{attribute 'GeneratedUsingTerminal: EK1100-0000-0018'}
{attribute addProperty BoxType "EK1100-0000-0018"}
{attribute addProperty Id "Beckhoff_EJ7xxxEK1122Beckhoff_EJ7xxxEK1122_3A43B2222A_0001_EJ7031_0000_0026EJ7031_31AD1E8938A_0002_EJ7037_0000_0020EJ7037_B6E6359B46A_0003_EJ7041_0052_0016EJ7041_31AD1E8938A_0004_EJ7047_0000_0018EJ7047_B6E6359B46A_0005_EJ7047_0000_0019EJ7047_B6E6359B46A_0006_EJ7047_0000_0020EJ7047_B6E6359B46A_0007_EJ7342_0000_0019EJ7342_A970B60778A_0008_EJ7342_0000_0020EJ7342_A970B60778A_0009_EJ7211_0010_0026EJ7211_91DE43F025A_0010_EJ7211_0010_0027EJ7211_91DE43F025A_0011_EJ7211_0010_0028EJ7211_91DE43F025A_0012_EJ7211_0010_0029EJ7211_91DE43F025A_0013_EJ7211_0010_0030EJ7211_0985306B26A_0014_EJ7211_0010_0031EJ7211_0985306B26A_0015_EJ7211_0010_0032EJ7211_0985306B26A_0016_EJ7211_0011_0026EJ7211_24495B2825A_0017_EJ7211_0011_0027EJ7211_24495B2825A_0018_EJ7211_0011_0028EJ7211_24495B2825A_0019_EJ7211_0011_0029EJ7211_24495B2825A_0020_EJ7211_0011_0030EJ7211_24495B2825A_0021_EJ7211_0011_0031EJ7211_24495B2825A_0022_EJ7211_0011_0032EJ7211_24495B2825A_0023_EJ7211_9414_0029EJ7211_91DE43F025A_0024_EJ7211_9414_0030EJ7211_49D18A3927A_0025_EJ7211_9414_0031EJ7211_49D18A3927A_0026_EJ7211_9414_0032EJ7211_49D18A3927A_0027_EJ7211_9415_0029EJ7211_24495B2825A_0028_EJ7211_9415_0030EJ7211_24495B2825A_0029_EJ7211_9415_0031EJ7211_24495B2825A_0030_EJ7211_9415_0032EJ7211_24495B2825A_0031_EJ7334_0008_0016EJ7334_074992E952A_0032_EJ7411_0000_0018EJ7411_D6A8D49830"}
{attribute addProperty CRC "2174237961"}
{attribute addProperty Size "1059"}
TYPE Beckhoff_EJ7xxx_81983D09 EXTENDS EK1100_1FC0878B :
STRUCT
	{attribute addProperty Name "Beckhoff_EJ7xxxEK1122"}
	{attribute addProperty PreviousPort "Beckhoff EJ7xxx : B"}
	Beckhoff_EJ7xxxEK1122 : Beckhoff_EJ7xxxEK1122_3A43B222;
	{attribute addProperty Name "A_0001_EJ7031_0000_0026"}
	{attribute addProperty PreviousPort "Beckhoff EJ7xxxEK1122 : C"}
	A_0001_EJ7031_0000_0026 : EJ7031_31AD1E89;
	{attribute addProperty Name "A_0002_EJ7037_0000_0020"}
	{attribute addProperty PreviousPort "A_0001(EJ7031-0000-0026) : B"}
	A_0002_EJ7037_0000_0020 : EJ7037_B6E6359B;
	{attribute addProperty Name "A_0003_EJ7041_0052_0016"}
	{attribute addProperty PreviousPort "A_0002(EJ7037-0000-0020) : B"}
	A_0003_EJ7041_0052_0016 : EJ7041_31AD1E89;
	{attribute addProperty Name "A_0004_EJ7047_0000_0018"}
	{attribute addProperty PreviousPort "A_0003(EJ7041-0052-0016) : B"}
	A_0004_EJ7047_0000_0018 : EJ7047_B6E6359B;
	{attribute addProperty Name "A_0005_EJ7047_0000_0019"}
	{attribute addProperty PreviousPort "A_0004(EJ7047-0000-0018) : B"}
	A_0005_EJ7047_0000_0019 : EJ7047_B6E6359B;
	{attribute addProperty Name "A_0006_EJ7047_0000_0020"}
	{attribute addProperty PreviousPort "A_0005(EJ7047-0000-0019) : B"}
	A_0006_EJ7047_0000_0020 : EJ7047_B6E6359B;
	{attribute addProperty Name "A_0007_EJ7342_0000_0019"}
	{attribute addProperty PreviousPort "A_0006(EJ7047-0000-0020) : B"}
	A_0007_EJ7342_0000_0019 : EJ7342_A970B607;
	{attribute addProperty Name "A_0008_EJ7342_0000_0020"}
	{attribute addProperty PreviousPort "A_0007(EJ7342-0000-0019) : B"}
	A_0008_EJ7342_0000_0020 : EJ7342_A970B607;
	{attribute addProperty Name "A_0009_EJ7211_0010_0026"}
	{attribute addProperty PreviousPort "A_0008(EJ7342-0000-0020) : B"}
	A_0009_EJ7211_0010_0026 : EJ7211_91DE43F0;
	{attribute addProperty Name "A_0010_EJ7211_0010_0027"}
	{attribute addProperty PreviousPort "A_0009(EJ7211-0010-0026) : B"}
	A_0010_EJ7211_0010_0027 : EJ7211_91DE43F0;
	{attribute addProperty Name "A_0011_EJ7211_0010_0028"}
	{attribute addProperty PreviousPort "A_0010(EJ7211-0010-0027) : B"}
	A_0011_EJ7211_0010_0028 : EJ7211_91DE43F0;
	{attribute addProperty Name "A_0012_EJ7211_0010_0029"}
	{attribute addProperty PreviousPort "A_0011(EJ7211-0010-0028) : B"}
	A_0012_EJ7211_0010_0029 : EJ7211_91DE43F0;
	{attribute addProperty Name "A_0013_EJ7211_0010_0030"}
	{attribute addProperty PreviousPort "A_0012(EJ7211-0010-0029) : B"}
	A_0013_EJ7211_0010_0030 : EJ7211_0985306B;
	{attribute addProperty Name "A_0014_EJ7211_0010_0031"}
	{attribute addProperty PreviousPort "A_0013(EJ7211-0010-0030) : B"}
	A_0014_EJ7211_0010_0031 : EJ7211_0985306B;
	{attribute addProperty Name "A_0015_EJ7211_0010_0032"}
	{attribute addProperty PreviousPort "A_0014(EJ7211-0010-0031) : B"}
	A_0015_EJ7211_0010_0032 : EJ7211_0985306B;
	{attribute addProperty Name "A_0016_EJ7211_0011_0026"}
	{attribute addProperty PreviousPort "A_0015(EJ7211-0010-0032) : B"}
	A_0016_EJ7211_0011_0026 : EJ7211_24495B28;
	{attribute addProperty Name "A_0017_EJ7211_0011_0027"}
	{attribute addProperty PreviousPort "A_0016(EJ7211-0011-0026) : B"}
	A_0017_EJ7211_0011_0027 : EJ7211_24495B28;
	{attribute addProperty Name "A_0018_EJ7211_0011_0028"}
	{attribute addProperty PreviousPort "A_0017(EJ7211-0011-0027) : B"}
	A_0018_EJ7211_0011_0028 : EJ7211_24495B28;
	{attribute addProperty Name "A_0019_EJ7211_0011_0029"}
	{attribute addProperty PreviousPort "A_0018(EJ7211-0011-0028) : B"}
	A_0019_EJ7211_0011_0029 : EJ7211_24495B28;
	{attribute addProperty Name "A_0020_EJ7211_0011_0030"}
	{attribute addProperty PreviousPort "A_0019(EJ7211-0011-0029) : B"}
	A_0020_EJ7211_0011_0030 : EJ7211_24495B28;
	{attribute addProperty Name "A_0021_EJ7211_0011_0031"}
	{attribute addProperty PreviousPort "A_0020(EJ7211-0011-0030) : B"}
	A_0021_EJ7211_0011_0031 : EJ7211_24495B28;
	{attribute addProperty Name "A_0022_EJ7211_0011_0032"}
	{attribute addProperty PreviousPort "A_0021(EJ7211-0011-0031) : B"}
	A_0022_EJ7211_0011_0032 : EJ7211_24495B28;
	{attribute addProperty Name "A_0023_EJ7211_9414_0029"}
	{attribute addProperty PreviousPort "A_0022(EJ7211-0011-0032) : B"}
	A_0023_EJ7211_9414_0029 : EJ7211_91DE43F0;
	{attribute addProperty Name "A_0024_EJ7211_9414_0030"}
	{attribute addProperty PreviousPort "A_0023(EJ7211-9414-0029) : B"}
	A_0024_EJ7211_9414_0030 : EJ7211_49D18A39;
	{attribute addProperty Name "A_0025_EJ7211_9414_0031"}
	{attribute addProperty PreviousPort "A_0024(EJ7211-9414-0030) : B"}
	A_0025_EJ7211_9414_0031 : EJ7211_49D18A39;
	{attribute addProperty Name "A_0026_EJ7211_9414_0032"}
	{attribute addProperty PreviousPort "A_0025(EJ7211-9414-0031) : B"}
	A_0026_EJ7211_9414_0032 : EJ7211_49D18A39;
	{attribute addProperty Name "A_0027_EJ7211_9415_0029"}
	{attribute addProperty PreviousPort "A_0026(EJ7211-9414-0032) : B"}
	A_0027_EJ7211_9415_0029 : EJ7211_24495B28;
	{attribute addProperty Name "A_0028_EJ7211_9415_0030"}
	{attribute addProperty PreviousPort "A_0027(EJ7211-9415-0029) : B"}
	A_0028_EJ7211_9415_0030 : EJ7211_24495B28;
	{attribute addProperty Name "A_0029_EJ7211_9415_0031"}
	{attribute addProperty PreviousPort "A_0028(EJ7211-9415-0030) : B"}
	A_0029_EJ7211_9415_0031 : EJ7211_24495B28;
	{attribute addProperty Name "A_0030_EJ7211_9415_0032"}
	{attribute addProperty PreviousPort "A_0029(EJ7211-9415-0031) : B"}
	A_0030_EJ7211_9415_0032 : EJ7211_24495B28;
	{attribute addProperty Name "A_0031_EJ7334_0008_0016"}
	{attribute addProperty PreviousPort "A_0030(EJ7211-9415-0032) : B"}
	A_0031_EJ7334_0008_0016 : EJ7334_074992E9;
	{attribute addProperty Name "A_0032_EJ7411_0000_0018"}
	{attribute addProperty PreviousPort "A_0031(EJ7334-0008-0016) : B"}
	A_0032_EJ7411_0000_0018 : EJ7411_D6A8D498;
END_STRUCT
END_TYPE

(* stored: Version 1.2.0.0, ProductVersion 3.1.4024.9
   DUT Beckhoff_EJ7xxx_81983D09: Id {09822d5d-79fa-4fe4-97ef-f5e0e0733d4b} *)
